{attribute 'linkalways'} 
{attribute 'no_explicit_call' := 'This FB is a CLASS and must be accessed using methods or properties'}
{attribute 'enable_dynamic_creation'}
FUNCTION_BLOCK Node_F_VN_PutLabel EXTENDS Node
VAR
    sText : _STRING('');
    ipDestImage : _ITcVnImage;
    nX : _UDINT(1);
    nY : _UDINT(1);
    fFontScale : _LREAL(1.0);
    hrPrev : _HRESULT(S_OK);
	hresult : _HRESULT(S_OK);
END_VAR

METHOD PUBLIC  Clone : I_Node
VAR
	pNode : POINTER TO Node_F_VN_PutLabel;
END_VAR
pNode := __NEW(Node_F_VN_PutLabel);
Clone := pNode^;
END_METHOD

METHOD FB_init : BOOL
VAR_INPUT
	bInitRetains : BOOL; // if TRUE, the retain variables are initialized (warm start / cold start)
	bInCopyCode : BOOL;  // if TRUE, the instance afterwards gets moved into the copy code (online change)
END_VAR
AddInput('sText', sText);
AddInput('ipDestImage', ipDestImage);
AddInput('hrPrev', hrPrev);
AddOutput('ipDestImage', ipDestImage);
AddOutput('hresult',hresult);
AddParameter('nX', nX);
AddParameter('nY', nY);
AddParameter('fFontScale', fFontScale);
END_METHOD

METHOD PROTECTED  OnExecute : HRESULT
hresult.Value := F_VN_PutLabel(
    sText := sText.Value,
	ipDestImage := ipDestImage.Value,
	nX:= nX.Value,
	nY:= nY.Value,
    fFontScale := fFontScale.Value,
	hrPrev:= hrPrev.Value);
END_METHOD

END_FUNCTION_BLOCK

(* stored: Version 1.1.0.1, ProductVersion 3.1.4024.13
   POU Node_F_VN_PutLabel: Id {3fefe494-7bd2-06f6-3fd7-a98cb0ae54f9}, SpecialFunc None
   Folder Constructor: Id {9fde9761-c63d-09e6-25b6-8c435bf7b666}
   Method Clone: Id {ca80b2e9-03de-02d8-31ba-682a5d8e01e9}
   Method FB_init: Id {c856191b-c335-070f-034d-f200a0c45f74}
   Method OnExecute: Id {9b50e28c-bdf9-0083-1dd5-f384f949c647} *)
